(* Logix 5000 project; controller KTC_WT vendor 1 type 14 code 150 rev 30.11; software revision 30.00 *)

TASK MainTask (continuous, watchdog 500 ms) : MainProgram

MODULES
   Local : vendor 1 type 14 code 150 (Compact 0, rev 30.11)
      Counters : Embedded (Compact 3, rev 1.1, Output RPI 20 ms)
      Discrete_IO : Embedded (Compact 1, rev 3.1, Output RPI 20 ms)
      Analog_IO : Embedded (Compact 2, rev 1.1, Output RPI 80 ms)
END_MODULES

PROGRAM MainProgram   (* main routine MainRoutine *)
VAR
   H_1 : ALIAS FOR Local:1:O.Data.7;   // HEATER
   IR_1 : ALIAS FOR Local:1:I.Data.0;   // CUP POSITION SENSOR 1
   IR_2 : ALIAS FOR Local:1:I.Data.1;   // CUP POSITION SENSOR 2
   M_1 : ALIAS FOR Local:1:O.Data.5;   // PUMP
   M_2 : ALIAS FOR Local:1:O.Data.6;   // CONVEYER
   MAIN_SCALED : REAL;
   MAIN_SLOPE : REAL;
   PB_1 : BOOL;   // FILL TANK 1 BUTTON
   PB_2 : BOOL;   // FILL TANK 2 BUTTON
   PB_3 : BOOL;   // DROP WATER FROM TANK 1 BUTTON
   PB_4 : BOOL;   // DROP WATER FROM TANK 1 BUTTON
   PB_5 : BOOL;   // MOVE CONVEYER
   PB_6 : BOOL;   // HEATER
   RAW_MAIN : DINT;
   RAW_T1 : DINT;
   RAW_T2 : DINT;
   RAW_TEMP : DINT;
   SOL_1 : ALIAS FOR Local:1:O.Data.0;   // FILL TANK 1
   SOL_2 : ALIAS FOR Local:1:O.Data.1;   // FILL TANK 2
   SOL_3 : ALIAS FOR Local:1:O.Data.2;   // DROP 1
   SOL_4 : ALIAS FOR Local:1:O.Data.3;   // DROP 2
   SW_1 : BOOL;   // MANUAL/AUTO
   T1_SCALED : REAL;
   T1_SLOPE : REAL;
   T2_SCALED : REAL;
   T2_SLOPE : REAL;
   TEMP_SCALED : REAL;
   TEMP_SLOPE : REAL;
END_VAR

ROUTINE AUTO   (* ladder *)
END_ROUTINE

ROUTINE MainRoutine   (* ladder *)
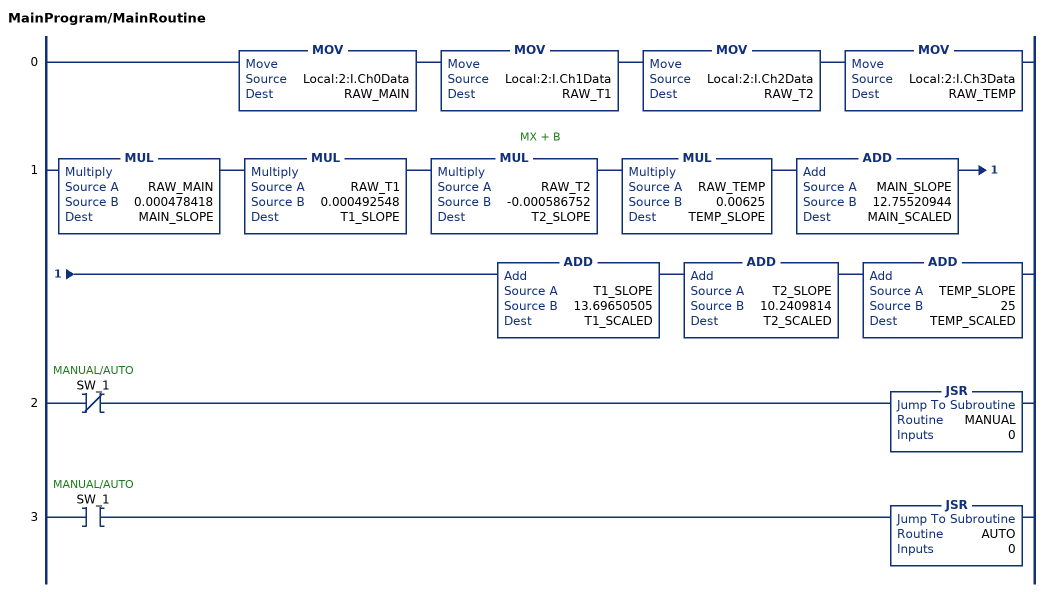
   0: MOV(Local:2:I.Ch0Data,RAW_MAIN)MOV(Local:2:I.Ch1Data,RAW_T1)MOV(Local:2:I.Ch2Data,RAW_T2)MOV(Local:2:I.Ch3Data,RAW_TEMP);
   // MX + B
   1: MUL(RAW_MAIN,0.000478418,MAIN_SLOPE)MUL(RAW_T1,0.000492548,T1_SLOPE)MUL(RAW_T2,-0.000586752,T2_SLOPE)MUL(RAW_TEMP,0.00625,TEMP_SLOPE)ADD(MAIN_SLOPE,12.75520944,MAIN_SCALED)ADD(T1_SLOPE,13.69650505,T1_SCALED)ADD(T2_SLOPE,10.2409814,T2_SCALED)ADD(TEMP_SLOPE,25,TEMP_SCALED);
   2: XIO(SW_1)JSR(MANUAL,0);
   3: XIC(SW_1)JSR(AUTO,0);
END_ROUTINE

ROUTINE MANUAL   (* ladder *)
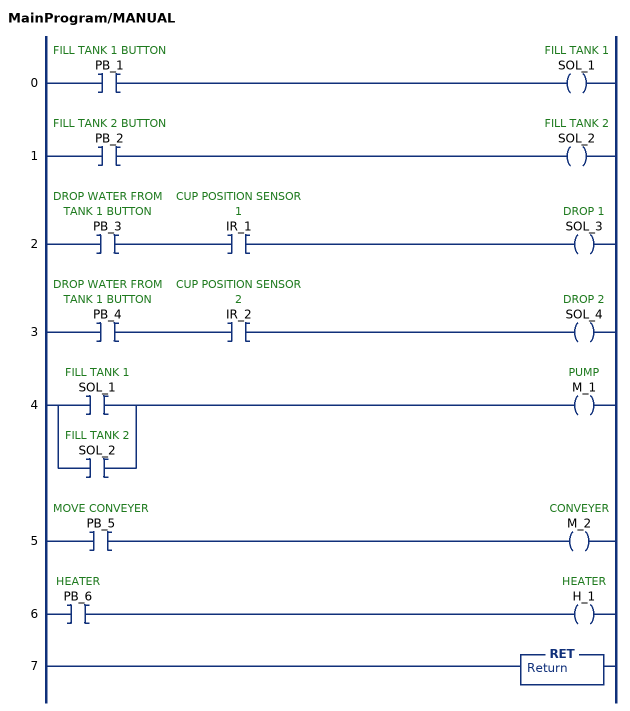
   0: XIC(PB_1)OTE(SOL_1);
   1: XIC(PB_2)OTE(SOL_2);
   2: XIC(PB_3)XIC(IR_1)OTE(SOL_3);
   3: XIC(PB_4)XIC(IR_2)OTE(SOL_4);
   4: [XIC(SOL_1) ,XIC(SOL_2) ]OTE(M_1);
   5: XIC(PB_5)OTE(M_2);
   6: XIC(PB_6)OTE(H_1);
   7: RET();
END_ROUTINE
END_PROGRAM
